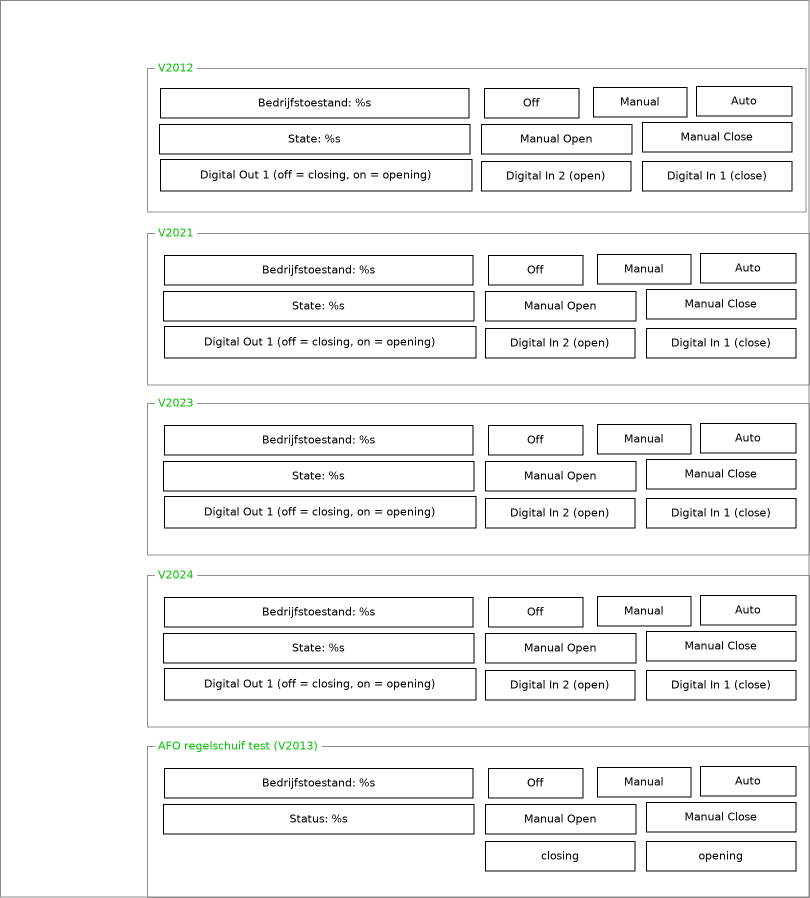
VISUALIZATION Visualization  // 810x898
    GroupBox (147,225 663x160), "V2021"
        RoundedRectangle (338,103 150x30), "Digital In 2 (open)", colour toggle: MAIN.digIn_V2021_2.internalState
            OnMouseDown: toggle MAIN.digIn_V2021_2.internalState
        RoundedRectangle (16,66 311x30), "State: %s", text variable: MAIN.V2021.currentState
        RoundedRectangle (17,30 309x30), "Bedrijfstoestand: %s", text variable: MAIN.V2021.currentMode
        RoundedRectangle (450,29 94x30), "Manual"
            OnMouseDown: execute { MAIN.V2021.currentMode := E_Bedrijfstoestand.manual; }
        RoundedRectangle (553,28 96x30), "Auto"
            OnMouseDown: execute { MAIN.V2021.currentMode := E_Bedrijfstoestand.auto; }
        RoundedRectangle (17,101 312x32), "Digital Out 1 (off = closing, on = opening)", colour toggle: MAIN.digOut_V2021.internalState
        RoundedRectangle (338,66 151x30), "Manual Open"
            OnMouseDown: execute { MAIN.V2021.manOpen := TRUE; }
        RoundedRectangle (499,64 150x30), "Manual Close"
            OnMouseDown: execute { MAIN.V2021.manClose := TRUE; }
        RoundedRectangle (499,103 150x30), "Digital In 1 (close)", colour toggle: MAIN.digIn_V2021_1.internalState
            OnMouseDown: toggle MAIN.digIn_V2021_1.internalState
        RoundedRectangle (341,30 95x30), "Off"
            OnMouseDown: execute { MAIN.V2021.currentMode := E_Bedrijfstoestand.off; }
    GroupBox (147,60 659x152), "V2012"
        RoundedRectangle (334,101 150x30), "Digital In 2 (open)", colour toggle: MAIN.digIn_V2012_2.internalState
            OnMouseDown: toggle MAIN.digIn_V2012_2.internalState
        RoundedRectangle (12,64 311x30), "State: %s", text variable: MAIN.V2012.currentState
        RoundedRectangle (13,28 309x30), "Bedrijfstoestand: %s", text variable: MAIN.V2012.currentMode
        RoundedRectangle (446,27 94x30), "Manual"
            OnMouseDown: execute { MAIN.V2012.currentMode := E_Bedrijfstoestand.manual; }
        RoundedRectangle (549,26 96x30), "Auto"
            OnMouseDown: execute { MAIN.V2012.currentMode := E_Bedrijfstoestand.auto; }
        RoundedRectangle (13,99 312x32), "Digital Out 1 (off = closing, on = opening)", colour toggle: MAIN.digOut_V2012.internalState
        RoundedRectangle (334,64 151x30), "Manual Open"
            OnMouseDown: execute { MAIN.V2012.manOpen := TRUE; }
        RoundedRectangle (495,62 150x30), "Manual Close"
            OnMouseDown: execute { MAIN.V2012.manClose := TRUE; }
        RoundedRectangle (495,101 150x30), "Digital In 1 (close)", colour toggle: MAIN.digIn_V2012_1.internalState
            OnMouseDown: toggle MAIN.digIn_V2012_1.internalState
        RoundedRectangle (337,28 95x30), "Off"
            OnMouseDown: execute { MAIN.V2012.currentMode := E_Bedrijfstoestand.off; }
    GroupBox (147,395 663x160), "V2023"
        RoundedRectangle (338,103 150x30), "Digital In 2 (open)", colour toggle: MAIN.digIn_V2023_2.internalState
            OnMouseDown: toggle MAIN.digIn_V2023_2.internalState
        RoundedRectangle (16,66 311x30), "State: %s", text variable: MAIN.V2023.currentState
        RoundedRectangle (17,30 309x30), "Bedrijfstoestand: %s", text variable: MAIN.V2023.currentMode
        RoundedRectangle (450,29 94x30), "Manual"
            OnMouseDown: execute { MAIN.V2023.currentMode := E_Bedrijfstoestand.manual; }
        RoundedRectangle (553,28 96x30), "Auto"
            OnMouseDown: execute { MAIN.V2023.currentMode := E_Bedrijfstoestand.auto; }
        RoundedRectangle (17,101 312x32), "Digital Out 1 (off = closing, on = opening)", colour toggle: MAIN.digOut_V2023.internalState
        RoundedRectangle (338,66 151x30), "Manual Open"
            OnMouseDown: execute { MAIN.V2023.manOpen := TRUE; }
        RoundedRectangle (499,64 150x30), "Manual Close"
            OnMouseDown: execute { MAIN.V2023.manClose := TRUE; }
        RoundedRectangle (499,103 150x30), "Digital In 1 (close)", colour toggle: MAIN.digIn_V2023_1.internalState
            OnMouseDown: toggle MAIN.digIn_V2023_1.internalState
        RoundedRectangle (341,30 95x30), "Off"
            OnMouseDown: execute { MAIN.V2023.currentMode := E_Bedrijfstoestand.off; }
    GroupBox (147,567 663x160), "V2024"
        RoundedRectangle (338,103 150x30), "Digital In 2 (open)", colour toggle: MAIN.digIn_V2024_2.internalState
            OnMouseDown: toggle MAIN.digIn_V2024_2.internalState
        RoundedRectangle (16,66 311x30), "State: %s", text variable: MAIN.V2024.currentState
        RoundedRectangle (17,30 309x30), "Bedrijfstoestand: %s", text variable: MAIN.V2024.currentMode
        RoundedRectangle (450,29 94x30), "Manual"
            OnMouseDown: execute { MAIN.V2024.currentMode := E_Bedrijfstoestand.manual; }
        RoundedRectangle (553,28 96x30), "Auto"
            OnMouseDown: execute { MAIN.V2024.currentMode := E_Bedrijfstoestand.auto; }
        RoundedRectangle (17,101 312x32), "Digital Out 1 (off = closing, on = opening)", colour toggle: MAIN.digOut_V2024.internalState
        RoundedRectangle (338,66 151x30), "Manual Open"
            OnMouseDown: execute { MAIN.V2024.manOpen := TRUE; }
        RoundedRectangle (499,64 150x30), "Manual Close"
            OnMouseDown: execute { MAIN.V2024.manClose := TRUE; }
        RoundedRectangle (499,103 150x30), "Digital In 1 (close)", colour toggle: MAIN.digIn_V2024_1.internalState
            OnMouseDown: toggle MAIN.digIn_V2024_1.internalState
        RoundedRectangle (341,30 95x30), "Off"
            OnMouseDown: execute { MAIN.V2024.currentMode := E_Bedrijfstoestand.off; }
    GroupBox (147,738 663x160), "AFO regelschuif test (V2013)", tooltip "niet final"
        RoundedRectangle (338,103 150x30), "closing", colour toggle: MAIN.V2013.outputClose
            OnMouseDown: toggle MAIN.digIn_V2024_2.internalState
        RoundedRectangle (16,66 311x30), "Status: %s", text variable: MAIN.V2013.currentState
        RoundedRectangle (17,30 309x30), "Bedrijfstoestand: %s", text variable: MAIN.V2013.currentMode
        RoundedRectangle (450,29 94x30), "Manual"
            OnMouseDown: execute { MAIN.V2024.currentMode := E_Bedrijfstoestand.manual; }
        RoundedRectangle (553,28 96x30), "Auto"
            OnMouseDown: execute { MAIN.V2024.currentMode := E_Bedrijfstoestand.auto; }
        RoundedRectangle (499,64 150x30), "Manual Close"
            OnMouseDown: execute { MAIN.V2024.manClose := TRUE; }
        RoundedRectangle (499,103 150x30), "opening", colour toggle: MAIN.V2013.outputOpen
            OnMouseDown: toggle MAIN.digIn_V2024_1.internalState
        RoundedRectangle (341,30 95x30), "Off"
            OnMouseDown: execute { MAIN.V2024.currentMode := E_Bedrijfstoestand.off; }
        RoundedRectangle (338,66 151x30), "Manual Open"
            OnMouseDown: execute { MAIN.V2024.manOpen := TRUE; }
END_VISUALIZATION

(* stored: Version 1.1.0.1, ProductVersion 3.1.4026.8
   Visu Visualization: Id {cf74a335-0ba7-461e-8ba0-0c2c14956010} *)
